FUNCTION VecAdd : Vec3
VAR_INPUT
	a, b : Vec3;
END_VAR
VAR
	i : INT;
END_VAR

FOR i := 0 TO 2 DO
    VecAdd.data[i] := a.data[i] + b.data[i]; 
END_FOR

END_FUNCTION

(* stored: Version 1.1.0.1, ProductVersion 3.1.4024.2
   POU VecAdd: Id {9a38d8a7-f9a5-4b94-a045-01f1cfce1efb}, SpecialFunc None *)
